        $ 646 "subir≔pose_sub(get_actual_tcp_pose(), bajada_broca)"
        global subir= pose_sub ( get_actual_tcp_pose (), bajada_broca)
        $ 647 "subir" "breakAfter"
        movel(subir, a=0.01, v=0.005)
        $ 648 "bajada_broca≔pose_sub(bajada_broca, bajada)"
        global bajada_broca= pose_sub (bajada_broca, bajada)
        Loop_42 = Loop_42 + 1
      end
      $ 649 "Direction: Base Z+"
      global move_thread_flag_649=0
      thread move_thread_649():
        enter_critical
        move_thread_flag_649 = 1
        local towardsPos=calculate_point_to_move_towards(p[0.0,0.0,0.0,0.0,0.0,0.0], [0.0,0.0,1.0], 0.06)
        movel(towardsPos, a=0.035, v=0.03)
        move_thread_flag_649 = 2
        exit_critical
      end
      move_thread_flag_649 = 0
      move_thread_han_649 = run move_thread_649()
      while (True):
        sleep(1.0E-10)
        if (move_thread_flag_649 > 1):
          join move_thread_han_649
          $ 650 "Until (distance)"
          break
        end
        sync()
      end
      $ 651 "Set CO[1]=Apagar"
      set_configurable_digital_out(1, False)
      $ 652 "barreno_actual≔barreno_actual+1"
      global barreno_actual=barreno_actual+1
      $ 653 "Call Quitar_broca"
      Quitar_broca()
      $ 654 "Call Poner_broca"
      Poner_broca()
    end
    $ 655 "EF"
    $ 656 "'desbaste_inicial'"
    # 'desbaste_inicial'
    $ 657 "bajada_broca≔p[0,0,-0.012,0,0,0]"
    global bajada_broca=p[0,0,-0.012,0,0,0]
    $ 658 "barrenos_menos1≔9"
    global barrenos_menos1=9
    $ 659 "barreno_actual≔0"
    global barreno_actual=0
    $ 660 "Loop barreno_actual≤barrenos_menos1"
    while (barreno_actual <= barrenos_menos1):
      $ 661 "Perforacion"
      $ 662 "MoveL"
      $ 663 "internos≔interpolate_pose(Linea2_E, Linea2_F, barreno_actual/barrenos_menos1)"
      global internos= interpolate_pose (Linea2_E_p, Linea2_F_p, barreno_actual/barrenos_menos1)
      $ 664 "internos" "breakAfter"
      movel(internos, a=0.5, v=0.1)
      $ 665 "'desbaste_inicial'"
      # 'desbaste_inicial'
      $ 666 "bajada_broca≔p[0,0,-0.012,0,0,0]"
      global bajada_broca=p[0,0,-0.012,0,0,0]
      $ 667 "bajada≔p[0,0,0.012,0,0,0]"
      global bajada=p[0,0,0.012,0,0,0]
      $ 668 "Direction: Base Z-"
      global move_thread_flag_668=0
      thread move_thread_668():
        enter_critical
        move_thread_flag_668 = 1
        local towardsPos=calculate_point_to_move_towards(p[0.0,0.0,0.0,0.0,0.0,0.0], [0.0,0.0,-1.0], 0.055)
        movel(towardsPos, a=0.025, v=0.02)
        move_thread_flag_668 = 2
        exit_critical
      end
      move_thread_flag_668 = 0
      move_thread_han_668 = run move_thread_668()
      while (True):
        sleep(1.0E-10)
        if (move_thread_flag_668 > 1):
          join move_thread_han_668
          $ 669 "Until (distance)"
          break
        end
        sync()
      end
      $ 670 "Popup: punto contacto alanzdo"
      popup("punto contacto alanzdo", "Mensaje", False, False, blocking=True)
      $ 671 "Direction: Base Z+"
      global move_thread_flag_671=0
      thread move_thread_671():
        enter_critical
        move_thread_flag_671 = 1
        local towardsPos=calculate_point_to_move_towards(p[0.0,0.0,0.0,0.0,0.0,0.0], [0.0,0.0,1.0], 0.001)
        movel(towardsPos, a=0.005, v=0.003)
        move_thread_flag_671 = 2
        exit_critical
      end
      move_thread_flag_671 = 0
      move_thread_han_671 = run move_thread_671()
      while (True):
        sleep(1.0E-10)
        if (move_thread_flag_671 > 1):
          join move_thread_han_671
          $ 672 "Until (distance)"
          break
        end
        sync()
      end
      $ 673 "Wait: 0.3"
      sleep(0.3)
      $ 674 "Set CO[1]=Encender"
      set_configurable_digital_out(1, True)
      $ 675 "Wait: 0.3"
      sleep(0.3)
      $ 676 "Loop 2 times"
      Loop_44 = 0
      while (Loop_44 < 2):
        $ 677 "bajar≔pose_add(get_actual_tcp_pose(), bajada_broca)"
        global bajar= pose_add ( get_actual_tcp_pose (), bajada_broca)
        $ 678 "bajar" "breakAfter"
        movel(bajar, a=0.005, v=0.001)
        $ 679 "subir≔pose_sub(get_actual_tcp_pose(), bajada_broca)"
        global subir= pose_sub ( get_actual_tcp_pose (), bajada_broca)
        $ 680 "subir" "breakAfter"
        movel(subir, a=0.01, v=0.005)
        $ 681 "bajada_broca≔pose_sub(bajada_broca, bajada)"
        global bajada_broca= pose_sub (bajada_broca, bajada)
        Loop_44 = Loop_44 + 1
      end
      $ 682 "Direction: Base Z+"
      global move_thread_flag_682=0
      thread move_thread_682():
        enter_critical
        move_thread_flag_682 = 1
        local towardsPos=calculate_point_to_move_towards(p[0.0,0.0,0.0,0.0,0.0,0.0], [0.0,0.0,1.0], 0.06)
        movel(towardsPos, a=0.035, v=0.03)
        move_thread_flag_682 = 2
        exit_critical
      end
      move_thread_flag_682 = 0
      move_thread_han_682 = run move_thread_682()
      while (True):
        sleep(1.0E-10)
        if (move_thread_flag_682 > 1):
          join move_thread_han_682
          $ 683 "Until (distance)"
          break
        end
        sync()
      end
      $ 684 "Set CO[1]=Apagar"
      set_configurable_digital_out(1, False)
      $ 685 "barreno_actual≔barreno_actual+1"
      global barreno_actual=barreno_actual+1
      $ 686 "If barreno_actual>barrenos_menos1"
      if (barreno_actual>barrenos_menos1):
        $ 687 "cambiar_broca≔ True "
        global cambiar_broca=  True
      end
      $ 688 "Call Quitar_broca"
      Quitar_broca()
      $ 689 "Call Poner_broca"
      Poner_broca()
    end
    $ 690 "Popup: Linea2 con full Terminada!"
    popup("Linea2 con full Terminada!", "Mensaje", False, False, blocking=True)
    $ 691 "Posicion3"
    $ 692 "eje7≔3"
    global eje7=3
    $ 693 "Broca_1"
    $ 694 "Linea3"
    $ 695 "Marcar_puntos"
    $ 696 "MoveL"
    $ 697 "punto_inicio1" "breakAfter"
    movel(punto_inicio1_p, a=0.5, v=0.1)
    $ 698 "Linea3_A" "breakAfter"
    movel(Linea3_A_p, a=0.5, v=0.1)
    $ 699 "Linea3_B" "breakAfter"
    movel(Linea3_B_p, a=0.5, v=0.1)
    $ 700 "Linea3_C" "breakAfter"
    movel(Linea3_C_p, a=0.5, v=0.1)
    $ 701 "Linea3_D" "breakAfter"
    movel(Linea3_D_p, a=0.5, v=0.1)
    $ 702 "Linea3_E" "breakAfter"
    movel(Linea3_E_p, a=0.5, v=0.1)
    $ 703 "Linea3_F" "breakAfter"
    movel(Linea3_F_p, a=0.5, v=0.1)
    $ 704 "AB"
    $ 705 "'desbaste_inicial'"
    # 'desbaste_inicial'
    $ 706 "bajada_broca≔p[0,0,-0.008,0,0,0]"
    global bajada_broca=p[0,0,-0.008,0,0,0]
    $ 707 "barrenos_menos1≔8"
    global barrenos_menos1=8
    $ 708 "barreno_actual≔0"
    global barreno_actual=0
    $ 709 "Loop barreno_actual≤barrenos_menos1"
    while (barreno_actual <= barrenos_menos1):
      $ 710 "Perforacion"
      $ 711 "MoveL"
      $ 712 "internos≔interpolate_pose(Linea3_A, Linea3_B, barreno_actual/barrenos_menos1)"
      global internos= interpolate_pose (Linea3_A_p, Linea3_B_p, barreno_actual/barrenos_menos1)
      $ 713 "internos" "breakAfter"
      movel(internos, a=0.5, v=0.1)
      $ 714 "'desbaste_inicial'"
      # 'desbaste_inicial'
      $ 715 "bajada_broca≔p[0,0,-0.008,0,0,0]"
      global bajada_broca=p[0,0,-0.008,0,0,0]
      $ 716 "bajada≔p[0,0,0.008,0,0,0]"
      global bajada=p[0,0,0.008,0,0,0]
      $ 717 "Direction: Base Z-"
      global move_thread_flag_717=0
      thread move_thread_717():
        enter_critical
        move_thread_flag_717 = 1
        local towardsPos=calculate_point_to_move_towards(p[0.0,0.0,0.0,0.0,0.0,0.0], [0.0,0.0,-1.0], 0.055)
        movel(towardsPos, a=0.015, v=0.02)
        move_thread_flag_717 = 2
        exit_critical
      end
      move_thread_flag_717 = 0
      move_thread_han_717 = run move_thread_717()
      while (True):
        sleep(1.0E-10)
        if (move_thread_flag_717 > 1):
          join move_thread_han_717
          $ 718 "Until (distance)"
          break
        end
        sync()
      end
      $ 719 "Popup: punto contacto alanzdo"
      popup("punto contacto alanzdo", "Mensaje", False, False, blocking=True)
      $ 720 "Direction: Base Z+"
      global move_thread_flag_720=0
      thread move_thread_720():
        enter_critical
        move_thread_flag_720 = 1
        local towardsPos=calculate_point_to_move_towards(p[0.0,0.0,0.0,0.0,0.0,0.0], [0.0,0.0,1.0], 0.001)
        movel(towardsPos, a=0.005, v=0.003)
        move_thread_flag_720 = 2
        exit_critical
      end
      move_thread_flag_720 = 0
      move_thread_han_720 = run move_thread_720()
      while (True):
        sleep(1.0E-10)
        if (move_thread_flag_720 > 1):
          join move_thread_han_720
          $ 721 "Until (distance)"
          break
        end
        sync()
      end
      $ 722 "Wait: 0.3"
      sleep(0.3)
      $ 723 "Set CO[1]=Encender"
      set_configurable_digital_out(1, True)
      $ 724 "Wait: 0.3"
      sleep(0.3)
      $ 725 "Loop 3 times"
      Loop_26 = 0
      while (Loop_26 < 3):
        $ 726 "bajar≔pose_add(get_actual_tcp_pose(), bajada_broca)"
        global bajar= pose_add ( get_actual_tcp_pose (), bajada_broca)
        $ 727 "bajar" "breakAfter"
        movel(bajar, a=0.005, v=0.001)
        $ 728 "subir≔pose_sub(get_actual_tcp_pose(), bajada_broca)"
        global subir= pose_sub ( get_actual_tcp_pose (), bajada_broca)
        $ 729 "subir" "breakAfter"
        movel(subir, a=0.01, v=0.005)
        $ 730 "bajada_broca≔pose_sub(bajada_broca, bajada)"
        global bajada_broca= pose_sub (bajada_broca, bajada)
        Loop_26 = Loop_26 + 1
      end
      $ 731 "Direction: Base Z+"
      global move_thread_flag_731=0
      thread move_thread_731():
        enter_critical
        move_thread_flag_731 = 1
        local towardsPos=calculate_point_to_move_towards(p[0.0,0.0,0.0,0.0,0.0,0.0], [0.0,0.0,1.0], 0.06)
        movel(towardsPos, a=0.035, v=0.03)
        move_thread_flag_731 = 2
        exit_critical
      end
      move_thread_flag_731 = 0
      move_thread_han_731 = run move_thread_731()
      while (True):
        sleep(1.0E-10)
        if (move_thread_flag_731 > 1):
          join move_thread_han_731
          $ 732 "Until (distance)"
          break
        end
        sync()
      end
      $ 733 "Set CO[1]=Apagar"
      set_configurable_digital_out(1, False)
      $ 734 "barreno_actual≔barreno_actual+1"
      global barreno_actual=barreno_actual+1
      $ 735 "Call Quitar_broca"
      Quitar_broca()
      $ 736 "Call Poner_broca"
      Poner_broca()
    end
    $ 737 "CD"
    $ 738 "'desbaste_inicial'"
    # 'desbaste_inicial'
    $ 739 "bajada_broca≔p[0,0,-0.008,0,0,0]"
    global bajada_broca=p[0,0,-0.008,0,0,0]
    $ 740 "barrenos_menos1≔8"
    global barrenos_menos1=8
    $ 741 "barreno_actual≔0"
    global barreno_actual=0
    $ 742 "Loop barreno_actual≤barrenos_menos1"
    while (barreno_actual <= barrenos_menos1):
      $ 743 "Perforacion"
      $ 744 "MoveL"
      $ 745 "internos≔interpolate_pose(Linea3_C, Linea3_D, barreno_actual/barrenos_menos1)"
      global internos= interpolate_pose (Linea3_C_p, Linea3_D_p, barreno_actual/barrenos_menos1)
      $ 746 "internos" "breakAfter"
      movel(internos, a=0.5, v=0.1)
      $ 747 "'desbaste_inicial'"
      # 'desbaste_inicial'
      $ 748 "bajada_broca≔p[0,0,-0.008,0,0,0]"
      global bajada_broca=p[0,0,-0.008,0,0,0]
      $ 749 "bajada≔p[0,0,0.008,0,0,0]"
      global bajada=p[0,0,0.008,0,0,0]
      $ 750 "Direction: Base Z-"
      global move_thread_flag_750=0
      thread move_thread_750():
        enter_critical
        move_thread_flag_750 = 1
        local towardsPos=calculate_point_to_move_towards(p[0.0,0.0,0.0,0.0,0.0,0.0], [0.0,0.0,-1.0], 0.055)
        movel(towardsPos, a=0.02, v=0.015)
        move_thread_flag_750 = 2
        exit_critical
      end
      move_thread_flag_750 = 0
      move_thread_han_750 = run move_thread_750()
      while (True):
        sleep(1.0E-10)
        if (move_thread_flag_750 > 1):
          join move_thread_han_750
          $ 751 "Until (distance)"
          break
        end
        sync()
      end
      $ 752 "Popup: punto contacto alanzdo"
      popup("punto contacto alanzdo", "Mensaje", False, False, blocking=True)
      $ 753 "Direction: Base Z+"
      global move_thread_flag_753=0
      thread move_thread_753():
        enter_critical
        move_thread_flag_753 = 1
        local towardsPos=calculate_point_to_move_towards(p[0.0,0.0,0.0,0.0,0.0,0.0], [0.0,0.0,1.0], 0.001)
        movel(towardsPos, a=0.005, v=0.003)
        move_thread_flag_753 = 2
        exit_critical
      end
      move_thread_flag_753 = 0
      move_thread_han_753 = run move_thread_753()
      while (True):
        sleep(1.0E-10)
        if (move_thread_flag_753 > 1):
          join move_thread_han_753
          $ 754 "Until (distance)"
          break
        end
        sync()
      end
      $ 755 "Wait: 0.3"
      sleep(0.3)
      $ 756 "Set CO[1]=Encender"
      set_configurable_digital_out(1, True)
      $ 757 "Wait: 0.3"
      sleep(0.3)
      $ 758 "Loop 3 times"
      Loop_28 = 0
      while (Loop_28 < 3):
        $ 759 "bajar≔pose_add(get_actual_tcp_pose(), bajada_broca)"
        global bajar= pose_add ( get_actual_tcp_pose (), bajada_broca)
        $ 760 "bajar" "breakAfter"
        movel(bajar, a=0.005, v=0.001)
        $ 761 "subir≔pose_sub(get_actual_tcp_pose(), bajada_broca)"
        global subir= pose_sub ( get_actual_tcp_pose (), bajada_broca)
        $ 762 "subir" "breakAfter"
        movel(subir, a=0.01, v=0.005)
        $ 763 "bajada_broca≔pose_sub(bajada_broca, bajada)"
        global bajada_broca= pose_sub (bajada_broca, bajada)
        Loop_28 = Loop_28 + 1
      end
      $ 764 "Direction: Base Z+"
      global move_thread_flag_764=0
      thread move_thread_764():
        enter_critical
        move_thread_flag_764 = 1
        local towardsPos=calculate_point_to_move_towards(p[0.0,0.0,0.0,0.0,0.0,0.0], [0.0,0.0,1.0], 0.06)
        movel(towardsPos, a=0.035, v=0.03)
        move_thread_flag_764 = 2
        exit_critical
      end
      move_thread_flag_764 = 0
      move_thread_han_764 = run move_thread_764()
      while (True):
        sleep(1.0E-10)
        if (move_thread_flag_764 > 1):
          join move_thread_han_764
          $ 765 "Until (distance)"
          break
        end
        sync()
      end
      $ 766 "Set CO[1]=Apagar"
      set_configurable_digital_out(1, False)
      $ 767 "barreno_actual≔barreno_actual+1"
      global barreno_actual=barreno_actual+1
      $ 768 "Call Quitar_broca"
      Quitar_broca()
      $ 769 "Call Poner_broca"
      Poner_broca()
    end
    $ 770 "EF"
    $ 771 "'desbaste_inicial'"
    # 'desbaste_inicial'
    $ 772 "bajada_broca≔p[0,0,-0.008,0,0,0]"
    global bajada_broca=p[0,0,-0.008,0,0,0]
    $ 773 "barrenos_menos1≔9"
    global barrenos_menos1=9
    $ 774 "barreno_actual≔0"
    global barreno_actual=0
    $ 775 "Loop barreno_actual≤barrenos_menos1"
    while (barreno_actual <= barrenos_menos1):
      $ 776 "Perforacion"
      $ 777 "MoveL"
      $ 778 "internos≔interpolate_pose(Linea3_E, Linea3_F, barreno_actual/barrenos_menos1)"
      global internos= interpolate_pose (Linea3_E_p, Linea3_F_p, barreno_actual/barrenos_menos1)
      $ 779 "internos" "breakAfter"
      movel(internos, a=0.5, v=0.1)
      $ 780 "'desbaste_inicial'"
      # 'desbaste_inicial'
      $ 781 "bajada_broca≔p[0,0,-0.008,0,0,0]"
      global bajada_broca=p[0,0,-0.008,0,0,0]
      $ 782 "bajada≔p[0,0,0.008,0,0,0]"
      global bajada=p[0,0,0.008,0,0,0]
      $ 783 "Direction: Base Z-"
      global move_thread_flag_783=0
      thread move_thread_783():
        enter_critical
        move_thread_flag_783 = 1
        local towardsPos=calculate_point_to_move_towards(p[0.0,0.0,0.0,0.0,0.0,0.0], [0.0,0.0,-1.0], 0.055)
        movel(towardsPos, a=0.015, v=0.02)
        move_thread_flag_783 = 2
        exit_critical
      end
      move_thread_flag_783 = 0
      move_thread_han_783 = run move_thread_783()
      while (True):
        sleep(1.0E-10)
        if (move_thread_flag_783 > 1):
          join move_thread_han_783
          $ 784 "Until (distance)"
          break
        end
        sync()
      end
      $ 785 "Popup: punto contacto alanzdo"
      popup("punto contacto alanzdo", "Mensaje", False, False, blocking=True)
      $ 786 "Direction: Base Z+"
      global move_thread_flag_786=0
      thread move_thread_786():
        enter_critical
        move_thread_flag_786 = 1
        local towardsPos=calculate_point_to_move_towards(p[0.0,0.0,0.0,0.0,0.0,0.0], [0.0,0.0,1.0], 0.001)
        movel(towardsPos, a=0.005, v=0.003)
        move_thread_flag_786 = 2
        exit_critical
      end
      move_thread_flag_786 = 0
      move_thread_han_786 = run move_thread_786()
      while (True):
        sleep(1.0E-10)
        if (move_thread_flag_786 > 1):
          join move_thread_han_786
          $ 787 "Until (distance)"
          break
        end
        sync()
      end
      $ 788 "Wait: 0.3"
      sleep(0.3)
      $ 789 "Set CO[1]=Encender"
      set_configurable_digital_out(1, True)
      $ 790 "Wait: 0.3"
      sleep(0.3)
      $ 791 "Loop 3 times"
      Loop_30 = 0
      while (Loop_30 < 3):
        $ 792 "bajar≔pose_add(get_actual_tcp_pose(), bajada_broca)"
        global bajar= pose_add ( get_actual_tcp_pose (), bajada_broca)
        $ 793 "bajar" "breakAfter"
        movel(bajar, a=0.005, v=0.001)
        $ 794 "subir≔pose_sub(get_actual_tcp_pose(), bajada_broca)"
        global subir= pose_sub ( get_actual_tcp_pose (), bajada_broca)
        $ 795 "subir" "breakAfter"
        movel(subir, a=0.01, v=0.005)
        $ 796 "bajada_broca≔pose_sub(bajada_broca, bajada)"
        global bajada_broca= pose_sub (bajada_broca, bajada)
        Loop_30 = Loop_30 + 1
      end
      $ 797 "Direction: Base Z+"
      global move_thread_flag_797=0
      thread move_thread_797():
        enter_critical
        move_thread_flag_797 = 1
        local towardsPos=calculate_point_to_move_towards(p[0.0,0.0,0.0,0.0,0.0,0.0], [0.0,0.0,1.0], 0.06)
        movel(towardsPos, a=0.035, v=0.03)
        move_thread_flag_797 = 2
        exit_critical
      end
      move_thread_flag_797 = 0
      move_thread_han_797 = run move_thread_797()
      while (True):
        sleep(1.0E-10)
        if (move_thread_flag_797 > 1):
          join move_thread_han_797
          $ 798 "Until (distance)"
          break
        end
        sync()
      end
      $ 799 "Set CO[1]=Apagar"
      set_configurable_digital_out(1, False)
      $ 800 "barreno_actual≔barreno_actual+1"
      global barreno_actual=barreno_actual+1
      $ 801 "Call Quitar_broca"
      Quitar_broca()
      $ 802 "Call Poner_broca"
      Poner_broca()
    end
    $ 803 "Popup: Linea1 con chica Terminada!"
    popup("Linea1 con chica Terminada!", "Mensaje", False, False, blocking=True)
    $ 804 "Linea4"
    $ 805 "Marcar_puntos"
    $ 806 "MoveL"
    $ 807 "punto_inicio1" "breakAfter"
    movel(punto_inicio1_p, a=0.5, v=0.1)
    $ 808 "Linea4_A" "breakAfter"
    movel(Linea4_A_p, a=0.5, v=0.1)
    $ 809 "Linea4_B" "breakAfter"
    movel(Linea4_B_p, a=0.5, v=0.1)
    $ 810 "Linea4_C" "breakAfter"
    movel(Linea4_C_p, a=0.5, v=0.1)
    $ 811 "Linea4_D" "breakAfter"
    movel(Linea4_D_p, a=0.5, v=0.1)
    $ 812 "Linea4_E" "breakAfter"
    movel(Linea4_E_p, a=0.5, v=0.1)
    $ 813 "Linea4_F" "breakAfter"
    movel(Linea4_F_p, a=0.5, v=0.1)
    $ 814 "AB"
    $ 815 "'desbaste_inicial'"
    # 'desbaste_inicial'
    $ 816 "bajada_broca≔p[0,0,-0.008,0,0,0]"
    global bajada_broca=p[0,0,-0.008,0,0,0]
    $ 817 "barrenos_menos1≔8"
    global barrenos_menos1=8
    $ 818 "barreno_actual≔0"
    global barreno_actual=0
    $ 819 "Loop barreno_actual≤barrenos_menos1"
    while (barreno_actual <= barrenos_menos1):
      $ 820 "Perforacion"
      $ 821 "MoveL"
      $ 822 "internos≔interpolate_pose(Linea4_A, Linea4_B, barreno_actual/barrenos_menos1)"
      global internos= interpolate_pose (Linea4_A_p, Linea4_B_p, barreno_actual/barrenos_menos1)
      $ 823 "internos" "breakAfter"
      movel(internos, a=0.5, v=0.1)
      $ 824 "'desbaste_inicial'"
      # 'desbaste_inicial'
      $ 825 "bajada_broca≔p[0,0,-0.008,0,0,0]"
      global bajada_broca=p[0,0,-0.008,0,0,0]
      $ 826 "bajada≔p[0,0,0.008,0,0,0]"
      global bajada=p[0,0,0.008,0,0,0]
      $ 827 "Direction: Base Z-"
      global move_thread_flag_827=0
      thread move_thread_827():
        enter_critical
        move_thread_flag_827 = 1
        local towardsPos=calculate_point_to_move_towards(p[0.0,0.0,0.0,0.0,0.0,0.0], [0.0,0.0,-1.0], 0.055)
        movel(towardsPos, a=0.015, v=0.02)
        move_thread_flag_827 = 2
        exit_critical
      end
      move_thread_flag_827 = 0
      move_thread_han_827 = run move_thread_827()
      while (True):
        sleep(1.0E-10)
        if (move_thread_flag_827 > 1):
          join move_thread_han_827
          $ 828 "Until (distance)"
          break
        end
        sync()
      end
      $ 829 "Popup: punto contacto alanzdo"
      popup("punto contacto alanzdo", "Mensaje", False, False, blocking=True)
      $ 830 "Direction: Base Z+"
      global move_thread_flag_830=0
      thread move_thread_830():
        enter_critical
        move_thread_flag_830 = 1
        local towardsPos=calculate_point_to_move_towards(p[0.0,0.0,0.0,0.0,0.0,0.0], [0.0,0.0,1.0], 0.002)
        movel(towardsPos, a=0.005, v=0.003)
        move_thread_flag_830 = 2
        exit_critical
      end
      move_thread_flag_830 = 0
      move_thread_han_830 = run move_thread_830()
      while (True):
        sleep(1.0E-10)
        if (move_thread_flag_830 > 1):
          join move_thread_han_830
          $ 831 "Until (distance)"
          break
        end
        sync()
      end
      $ 832 "Wait: 0.3"
      sleep(0.3)
      $ 833 "Set CO[1]=Encender"
      set_configurable_digital_out(1, True)
      $ 834 "Wait: 0.3"
      sleep(0.3)
      $ 835 "Loop 3 times"
      Loop_32 = 0
      while (Loop_32 < 3):
        $ 836 "bajar≔pose_add(get_actual_tcp_pose(), bajada_broca)"
        global bajar= pose_add ( get_actual_tcp_pose (), bajada_broca)
        $ 837 "bajar" "breakAfter"
        movel(bajar, a=0.005, v=0.001)
        $ 838 "subir≔pose_sub(get_actual_tcp_pose(), bajada_broca)"
        global subir= pose_sub ( get_actual_tcp_pose (), bajada_broca)
        $ 839 "subir" "breakAfter"
        movel(subir, a=0.01, v=0.005)
        $ 840 "bajada_broca≔pose_sub(bajada_broca, bajada)"
        global bajada_broca= pose_sub (bajada_broca, bajada)
        Loop_32 = Loop_32 + 1
      end
      $ 841 "Direction: Base Z+"
      global move_thread_flag_841=0
      thread move_thread_841():
        enter_critical
        move_thread_flag_841 = 1
        local towardsPos=calculate_point_to_move_towards(p[0.0,0.0,0.0,0.0,0.0,0.0], [0.0,0.0,1.0], 0.06)
        movel(towardsPos, a=0.035, v=0.03)
        move_thread_flag_841 = 2
        exit_critical
      end
      move_thread_flag_841 = 0
      move_thread_han_841 = run move_thread_841()
      while (True):
        sleep(1.0E-10)
        if (move_thread_flag_841 > 1):
          join move_thread_han_841
          $ 842 "Until (distance)"
          break
        end
        sync()
      end
      $ 843 "Set CO[1]=Apagar"
      set_configurable_digital_out(1, False)
      $ 844 "barreno_actual≔barreno_actual+1"
      global barreno_actual=barreno_actual+1
    end
    $ 847 "CD"
    $ 848 "'desbaste_inicial'"
    # 'desbaste_inicial'
    $ 849 "bajada_broca≔p[0,0,-0.008,0,0,0]"
    global bajada_broca=p[0,0,-0.008,0,0,0]
    $ 850 "barrenos_menos1≔8"
    global barrenos_menos1=8
    $ 851 "barreno_actual≔0"
    global barreno_actual=0
    $ 852 "Loop barreno_actual≤barrenos_menos1"
    while (barreno_actual <= barrenos_menos1):
      $ 853 "Perforacion"
      $ 854 "MoveL"
      $ 855 "internos≔interpolate_pose(Linea4_C, Linea4_D, barreno_actual/barrenos_menos1)"
      global internos= interpolate_pose (Linea4_C_p, Linea4_D_p, barreno_actual/barrenos_menos1)
      $ 856 "internos" "breakAfter"
      movel(internos, a=0.5, v=0.1)
      $ 857 "'desbaste_inicial'"
      # 'desbaste_inicial'
      $ 858 "bajada_broca≔p[0,0,-0.008,0,0,0]"
      global bajada_broca=p[0,0,-0.008,0,0,0]
      $ 859 "bajada≔p[0,0,0.008,0,0,0]"
      global bajada=p[0,0,0.008,0,0,0]
      $ 860 "Direction: Base Z-"
      global move_thread_flag_860=0
      thread move_thread_860():
        enter_critical
        move_thread_flag_860 = 1
        local towardsPos=calculate_point_to_move_towards(p[0.0,0.0,0.0,0.0,0.0,0.0], [0.0,0.0,-1.0], 0.055)
        movel(towardsPos, a=0.015, v=0.02)
        move_thread_flag_860 = 2
        exit_critical
      end
      move_thread_flag_860 = 0
      move_thread_han_860 = run move_thread_860()
      while (True):
        sleep(1.0E-10)
        if (move_thread_flag_860 > 1):
          join move_thread_han_860
          $ 861 "Until (distance)"
          break
        end
        sync()
      end
      $ 862 "Popup: punto contacto alanzdo"
      popup("punto contacto alanzdo", "Mensaje", False, False, blocking=True)
      $ 863 "Direction: Base Z+"
      global move_thread_flag_863=0
      thread move_thread_863():
        enter_critical
        move_thread_flag_863 = 1
        local towardsPos=calculate_point_to_move_towards(p[0.0,0.0,0.0,0.0,0.0,0.0], [0.0,0.0,1.0], 0.002)
        movel(towardsPos, a=0.005, v=0.003)
        move_thread_flag_863 = 2
        exit_critical
      end
      move_thread_flag_863 = 0
      move_thread_han_863 = run move_thread_863()
      while (True):
        sleep(1.0E-10)
        if (move_thread_flag_863 > 1):
          join move_thread_han_863
          $ 864 "Until (distance)"
          break
        end
        sync()
      end
      $ 865 "Wait: 0.3"
      sleep(0.3)
      $ 866 "Set CO[1]=Encender"
      set_configurable_digital_out(1, True)
      $ 867 "Wait: 0.3"
      sleep(0.3)
      $ 868 "Loop 3 times"
      Loop_35 = 0
      while (Loop_35 < 3):
        $ 869 "bajar≔pose_add(get_actual_tcp_pose(), bajada_broca)"
        global bajar= pose_add ( get_actual_tcp_pose (), bajada_broca)
        $ 870 "bajar" "breakAfter"
        movel(bajar, a=0.005, v=0.001)
        $ 871 "subir≔pose_sub(get_actual_tcp_pose(), bajada_broca)"
        global subir= pose_sub ( get_actual_tcp_pose (), bajada_broca)
        $ 872 "subir" "breakAfter"
        movel(subir, a=0.01, v=0.005)
        $ 873 "bajada_broca≔pose_sub(bajada_broca, bajada)"
        global bajada_broca= pose_sub (bajada_broca, bajada)
        Loop_35 = Loop_35 + 1
      end
      $ 874 "Direction: Base Z+"
      global move_thread_flag_874=0
      thread move_thread_874():
        enter_critical
        move_thread_flag_874 = 1
        local towardsPos=calculate_point_to_move_towards(p[0.0,0.0,0.0,0.0,0.0,0.0], [0.0,0.0,1.0], 0.06)
        movel(towardsPos, a=0.035, v=0.03)
        move_thread_flag_874 = 2
        exit_critical
      end
      move_thread_flag_874 = 0
      move_thread_han_874 = run move_thread_874()
      while (True):
        sleep(1.0E-10)
        if (move_thread_flag_874 > 1):
          join move_thread_han_874
          $ 875 "Until (distance)"
          break
        end
        sync()
      end
      $ 876 "Set CO[1]=Apagar"
      set_configurable_digital_out(1, False)
      $ 877 "barreno_actual≔barreno_actual+1"
      global barreno_actual=barreno_actual+1
    end
    $ 880 "EF"
    $ 881 "'desbaste_inicial'"
    # 'desbaste_inicial'
    $ 882 "bajada_broca≔p[0,0,-0.008,0,0,0]"
    global bajada_broca=p[0,0,-0.008,0,0,0]
    $ 883 "barrenos_menos1≔9"
    global barrenos_menos1=9
    $ 884 "barreno_actual≔0"
    global barreno_actual=0
    $ 885 "Loop barreno_actual≤barrenos_menos1"
    while (barreno_actual <= barrenos_menos1):
      $ 886 "Perforacion"
      $ 887 "MoveL"
      $ 888 "internos≔interpolate_pose(Linea4_E, Linea4_F, barreno_actual/barrenos_menos1)"
      global internos= interpolate_pose (Linea4_E_p, Linea4_F_p, barreno_actual/barrenos_menos1)
      $ 889 "internos" "breakAfter"
      movel(internos, a=0.5, v=0.1)
      $ 890 "'desbaste_inicial'"
      # 'desbaste_inicial'
      $ 891 "bajada_broca≔p[0,0,-0.008,0,0,0]"
      global bajada_broca=p[0,0,-0.008,0,0,0]
      $ 892 "bajada≔p[0,0,0.008,0,0,0]"
      global bajada=p[0,0,0.008,0,0,0]
      $ 893 "Direction: Base Z-"
      global move_thread_flag_893=0
      thread move_thread_893():
        enter_critical
        move_thread_flag_893 = 1
        local towardsPos=calculate_point_to_move_towards(p[0.0,0.0,0.0,0.0,0.0,0.0], [0.0,0.0,-1.0], 0.055)
        movel(towardsPos, a=0.015, v=0.02)
        move_thread_flag_893 = 2
        exit_critical
      end
      move_thread_flag_893 = 0
      move_thread_han_893 = run move_thread_893()
      while (True):
        sleep(1.0E-10)
        if (move_thread_flag_893 > 1):
          join move_thread_han_893
          $ 894 "Until (distance)"
          break
        end
        sync()
      end
      $ 895 "Popup: punto contacto alanzdo"
      popup("punto contacto alanzdo", "Mensaje", False, False, blocking=True)
      $ 896 "Direction: Base Z+"
      global move_thread_flag_896=0
      thread move_thread_896():
        enter_critical
        move_thread_flag_896 = 1
        local towardsPos=calculate_point_to_move_towards(p[0.0,0.0,0.0,0.0,0.0,0.0], [0.0,0.0,1.0], 0.002)
        movel(towardsPos, a=0.005, v=0.003)
        move_thread_flag_896 = 2
        exit_critical
      end
      move_thread_flag_896 = 0
      move_thread_han_896 = run move_thread_896()
      while (True):
        sleep(1.0E-10)
        if (move_thread_flag_896 > 1):
          join move_thread_han_896
          $ 897 "Until (distance)"
          break
        end
        sync()
      end
      $ 898 "Wait: 0.3"
      sleep(0.3)
      $ 899 "Set CO[1]=Encender"
      set_configurable_digital_out(1, True)
      $ 900 "Wait: 0.3"
      sleep(0.3)
      $ 901 "Loop 3 times"
      Loop_39 = 0
      while (Loop_39 < 3):
        $ 902 "bajar≔pose_add(get_actual_tcp_pose(), bajada_broca)"
        global bajar= pose_add ( get_actual_tcp_pose (), bajada_broca)
        $ 903 "bajar" "breakAfter"
        movel(bajar, a=0.005, v=0.001)
        $ 904 "subir≔pose_sub(get_actual_tcp_pose(), bajada_broca)"
        global subir= pose_sub ( get_actual_tcp_pose (), bajada_broca)
        $ 905 "subir" "breakAfter"
        movel(subir, a=0.01, v=0.005)
        $ 906 "bajada_broca≔pose_sub(bajada_broca, bajada)"
        global bajada_broca= pose_sub (bajada_broca, bajada)
        Loop_39 = Loop_39 + 1
      end
      $ 907 "Direction: Base Z+"
      global move_thread_flag_907=0
      thread move_thread_907():
        enter_critical
        move_thread_flag_907 = 1
        local towardsPos=calculate_point_to_move_towards(p[0.0,0.0,0.0,0.0,0.0,0.0], [0.0,0.0,1.0], 0.06)
        movel(towardsPos, a=0.035, v=0.03)
        move_thread_flag_907 = 2
        exit_critical
      end
      move_thread_flag_907 = 0
      move_thread_han_907 = run move_thread_907()
      while (True):
        sleep(1.0E-10)
        if (move_thread_flag_907 > 1):
          join move_thread_han_907
          $ 908 "Until (distance)"
          break
        end
        sync()
      end
      $ 909 "Set CO[1]=Apagar"
      set_configurable_digital_out(1, False)
      $ 910 "barreno_actual≔barreno_actual+1"
      global barreno_actual=barreno_actual+1
      $ 911 "If barreno_actual>barrenos_menos1"
      if (barreno_actual>barrenos_menos1):
        $ 912 "cambiar_broca≔ True "
        global cambiar_broca=  True
      end
    end
    $ 915 "Popup: Linea2 con chica Terminada!"
    popup("Linea2 con chica Terminada!", "Mensaje", False, False, blocking=True)
    $ 916 "Broca_2"
    $ 917 "Linea3"
    $ 918 "Marcar_puntos"
    $ 919 "MoveL"
    $ 920 "punto_inicio1" "breakAfter"
    movel(punto_inicio1_p, a=0.5, v=0.1)
    $ 921 "Linea3_A" "breakAfter"
    movel(Linea3_A_p, a=0.5, v=0.1)
    $ 922 "Linea3_B" "breakAfter"
    movel(Linea3_B_p, a=0.5, v=0.1)
    $ 923 "Linea3_C" "breakAfter"
    movel(Linea3_C_p, a=0.5, v=0.1)
    $ 924 "Linea3_D" "breakAfter"
    movel(Linea3_D_p, a=0.5, v=0.1)
    $ 925 "Linea3_E" "breakAfter"
    movel(Linea3_E_p, a=0.5, v=0.1)
    $ 926 "Linea3_F" "breakAfter"
    movel(Linea3_F_p, a=0.5, v=0.1)
    $ 927 "AB"
    $ 928 "'desbaste_inicial'"
    # 'desbaste_inicial'
    $ 929 "bajada_broca≔p[0,0,-0.012,0,0,0]"
    global bajada_broca=p[0,0,-0.012,0,0,0]
    $ 930 "barrenos_menos1≔8"
    global barrenos_menos1=8
    $ 931 "barreno_actual≔0"
    global barreno_actual=0
    $ 932 "Loop barreno_actual≤barrenos_menos1"
    while (barreno_actual <= barrenos_menos1):
      $ 933 "Perforacion"
      $ 934 "MoveL"
      $ 935 "internos≔interpolate_pose(Linea3_A, Linea3_B, barreno_actual/barrenos_menos1)"
      global internos= interpolate_pose (Linea3_A_p, Linea3_B_p, barreno_actual/barrenos_menos1)
      $ 936 "internos" "breakAfter"
      movel(internos, a=0.5, v=0.1)
      $ 937 "'desbaste_inicial'"
      # 'desbaste_inicial'
      $ 938 "bajada_broca≔p[0,0,-0.012,0,0,0]"
      global bajada_broca=p[0,0,-0.012,0,0,0]
      $ 939 "bajada≔p[0,0,0.012,0,0,0]"
      global bajada=p[0,0,0.012,0,0,0]
      $ 940 "Direction: Base Z-"
      global move_thread_flag_940=0
      thread move_thread_940():
        enter_critical
        move_thread_flag_940 = 1
        local towardsPos=calculate_point_to_move_towards(p[0.0,0.0,0.0,0.0,0.0,0.0], [0.0,0.0,-1.0], 0.055)
        movel(towardsPos, a=0.015, v=0.02)
        move_thread_flag_940 = 2
        exit_critical
      end
      move_thread_flag_940 = 0
      move_thread_han_940 = run move_thread_940()
      while (True):
        sleep(1.0E-10)
        if (move_thread_flag_940 > 1):
          join move_thread_han_940
          $ 941 "Until (distance)"
          break
        end
        sync()
      end
      $ 942 "Popup: punto contacto alanzdo"
      popup("punto contacto alanzdo", "Mensaje", False, False, blocking=True)
      $ 943 "Direction: Base Z+"
      global move_thread_flag_943=0
      thread move_thread_943():
        enter_critical
        move_thread_flag_943 = 1
        local towardsPos=calculate_point_to_move_towards(p[0.0,0.0,0.0,0.0,0.0,0.0], [0.0,0.0,1.0], 0.002)
        movel(towardsPos, a=0.005, v=0.003)
        move_thread_flag_943 = 2
        exit_critical
      end
      move_thread_flag_943 = 0
      move_thread_han_943 = run move_thread_943()
      while (True):
        sleep(1.0E-10)
        if (move_thread_flag_943 > 1):
          join move_thread_han_943
          $ 944 "Until (distance)"
          break
        end
        sync()
      end
      $ 945 "Wait: 0.3"
      sleep(0.3)
      $ 946 "Set CO[1]=Encender"
      set_configurable_digital_out(1, True)
      $ 947 "Wait: 0.3"
      sleep(0.3)
      $ 948 "Loop 2 times"
      Loop_70 = 0
      while (Loop_70 < 2):
        $ 949 "bajar≔pose_add(get_actual_tcp_pose(), bajada_broca)"
        global bajar= pose_add ( get_actual_tcp_pose (), bajada_broca)
        $ 950 "bajar" "breakAfter"
        movel(bajar, a=0.005, v=0.001)
        $ 951 "subir≔pose_sub(get_actual_tcp_pose(), bajada_broca)"
        global subir= pose_sub ( get_actual_tcp_pose (), bajada_broca)
        $ 952 "subir" "breakAfter"
        movel(subir, a=0.01, v=0.005)
        $ 953 "bajada_broca≔pose_sub(bajada_broca, bajada)"
        global bajada_broca= pose_sub (bajada_broca, bajada)
        Loop_70 = Loop_70 + 1
      end
      $ 954 "Direction: Base Z+"
      global move_thread_flag_954=0
      thread move_thread_954():
        enter_critical
        move_thread_flag_954 = 1
        local towardsPos=calculate_point_to_move_towards(p[0.0,0.0,0.0,0.0,0.0,0.0], [0.0,0.0,1.0], 0.06)
        movel(towardsPos, a=0.035, v=0.03)
        move_thread_flag_954 = 2
        exit_critical
      end
      move_thread_flag_954 = 0
      move_thread_han_954 = run move_thread_954()
      while (True):
        sleep(1.0E-10)
        if (move_thread_flag_954 > 1):
          join move_thread_han_954
          $ 955 "Until (distance)"
          break
        end
        sync()
      end
      $ 956 "Set CO[1]=Apagar"
      set_configurable_digital_out(1, False)
      $ 957 "barreno_actual≔barreno_actual+1"
      global barreno_actual=barreno_actual+1
    end
    $ 960 "CD"
    $ 961 "'desbaste_inicial'"
    # 'desbaste_inicial'
    $ 962 "bajada_broca≔p[0,0,-0.012,0,0,0]"
    global bajada_broca=p[0,0,-0.012,0,0,0]
    $ 963 "barrenos_menos1≔8"
    global barrenos_menos1=8
    $ 964 "barreno_actual≔0"
    global barreno_actual=0
    $ 965 "Loop barreno_actual≤barrenos_menos1"
    while (barreno_actual <= barrenos_menos1):
      $ 966 "Perforacion"
      $ 967 "MoveL"
      $ 968 "internos≔interpolate_pose(Linea3_C, Linea3_D, barreno_actual/barrenos_menos1)"
      global internos= interpolate_pose (Linea3_C_p, Linea3_D_p, barreno_actual/barrenos_menos1)
      $ 969 "internos" "breakAfter"
      movel(internos, a=0.5, v=0.1)
      $ 970 "'desbaste_inicial'"
      # 'desbaste_inicial'
      $ 971 "bajada_broca≔p[0,0,-0.012,0,0,0]"
      global bajada_broca=p[0,0,-0.012,0,0,0]
      $ 972 "bajada≔p[0,0,0.012,0,0,0]"
      global bajada=p[0,0,0.012,0,0,0]
      $ 973 "Direction: Base Z-"
      global move_thread_flag_973=0
      thread move_thread_973():
        enter_critical
        move_thread_flag_973 = 1
        local towardsPos=calculate_point_to_move_towards(p[0.0,0.0,0.0,0.0,0.0,0.0], [0.0,0.0,-1.0], 0.055)
        movel(towardsPos, a=0.02, v=0.015)
        move_thread_flag_973 = 2
        exit_critical
      end
      move_thread_flag_973 = 0
      move_thread_han_973 = run move_thread_973()
      while (True):
        sleep(1.0E-10)
        if (move_thread_flag_973 > 1):
          join move_thread_han_973
          $ 974 "Until (distance)"
          break
        end
        sync()
      end
      $ 975 "Popup: punto contacto alanzdo"
      popup("punto contacto alanzdo", "Mensaje", False, False, blocking=True)
      $ 976 "Direction: Base Z+"
      global move_thread_flag_976=0
      thread move_thread_976():
        enter_critical
        move_thread_flag_976 = 1
        local towardsPos=calculate_point_to_move_towards(p[0.0,0.0,0.0,0.0,0.0,0.0], [0.0,0.0,1.0], 0.002)
        movel(towardsPos, a=0.005, v=0.003)
        move_thread_flag_976 = 2
        exit_critical
      end
      move_thread_flag_976 = 0
      move_thread_han_976 = run move_thread_976()
      while (True):
        sleep(1.0E-10)
        if (move_thread_flag_976 > 1):
          join move_thread_han_976
          $ 977 "Until (distance)"
          break
        end
        sync()
      end
      $ 978 "Wait: 0.3"
      sleep(0.3)
      $ 979 "Set CO[1]=Encender"
      set_configurable_digital_out(1, True)
      $ 980 "Wait: 0.3"
      sleep(0.3)
      $ 981 "Loop 2 times"
      Loop_72 = 0
      while (Loop_72 < 2):
        $ 982 "bajar≔pose_add(get_actual_tcp_pose(), bajada_broca)"
        global bajar= pose_add ( get_actual_tcp_pose (), bajada_broca)
        $ 983 "bajar" "breakAfter"
        movel(bajar, a=0.005, v=0.001)
        $ 984 "subir≔pose_sub(get_actual_tcp_pose(), bajada_broca)"
        global subir= pose_sub ( get_actual_tcp_pose (), bajada_broca)
        $ 985 "subir" "breakAfter"
        movel(subir, a=0.01, v=0.005)
        $ 986 "bajada_broca≔pose_sub(bajada_broca, bajada)"
        global bajada_broca= pose_sub (bajada_broca, bajada)
        Loop_72 = Loop_72 + 1
      end
      $ 987 "Direction: Base Z+"
      global move_thread_flag_987=0
      thread move_thread_987():
        enter_critical
        move_thread_flag_987 = 1
        local towardsPos=calculate_point_to_move_towards(p[0.0,0.0,0.0,0.0,0.0,0.0], [0.0,0.0,1.0], 0.06)
        movel(towardsPos, a=0.035, v=0.03)
        move_thread_flag_987 = 2
        exit_critical
      end
      move_thread_flag_987 = 0
      move_thread_han_987 = run move_thread_987()
      while (True):
        sleep(1.0E-10)
        if (move_thread_flag_987 > 1):
          join move_thread_han_987
          $ 988 "Until (distance)"
          break
        end
        sync()
      end
      $ 989 "Set CO[1]=Apagar"
      set_configurable_digital_out(1, False)
      $ 990 "barreno_actual≔barreno_actual+1"
      global barreno_actual=barreno_actual+1
    end
    $ 993 "EF"
    $ 994 "'desbaste_inicial'"
    # 'desbaste_inicial'
    $ 995 "bajada_broca≔p[0,0,-0.012,0,0,0]"
    global bajada_broca=p[0,0,-0.012,0,0,0]
    $ 996 "barrenos_menos1≔9"
    global barrenos_menos1=9
    $ 997 "barreno_actual≔0"
    global barreno_actual=0
    $ 998 "Loop barreno_actual≤barrenos_menos1"
    while (barreno_actual <= barrenos_menos1):
      $ 999 "Perforacion"
      $ 1000 "MoveL"
      $ 1001 "internos≔interpolate_pose(Linea3_E, Linea3_F, barreno_actual/barrenos_menos1)"
      global internos= interpolate_pose (Linea3_E_p, Linea3_F_p, barreno_actual/barrenos_menos1)
      $ 1002 "internos" "breakAfter"
      movel(internos, a=0.5, v=0.1)
      $ 1003 "'desbaste_inicial'"
      # 'desbaste_inicial'
      $ 1004 "bajada_broca≔p[0,0,-0.012,0,0,0]"
      global bajada_broca=p[0,0,-0.012,0,0,0]
      $ 1005 "bajada≔p[0,0,0.012,0,0,0]"
      global bajada=p[0,0,0.012,0,0,0]
      $ 1006 "Direction: Base Z-"
      global move_thread_flag_1006=0
      thread move_thread_1006():
        enter_critical
        move_thread_flag_1006 = 1
        local towardsPos=calculate_point_to_move_towards(p[0.0,0.0,0.0,0.0,0.0,0.0], [0.0,0.0,-1.0], 0.055)
        movel(towardsPos, a=0.015, v=0.02)
        move_thread_flag_1006 = 2
        exit_critical
      end
      move_thread_flag_1006 = 0
      move_thread_han_1006 = run move_thread_1006()
      while (True):
        sleep(1.0E-10)
        if (move_thread_flag_1006 > 1):
          join move_thread_han_1006
          $ 1007 "Until (distance)"
          break
        end
        sync()
      end
      $ 1008 "Popup: punto contacto alanzdo"
      popup("punto contacto alanzdo", "Mensaje", False, False, blocking=True)
      $ 1009 "Direction: Base Z+"
      global move_thread_flag_1009=0
      thread move_thread_1009():
        enter_critical
        move_thread_flag_1009 = 1
        local towardsPos=calculate_point_to_move_towards(p[0.0,0.0,0.0,0.0,0.0,0.0], [0.0,0.0,1.0], 0.002)
        movel(towardsPos, a=0.005, v=0.003)
        move_thread_flag_1009 = 2
        exit_critical
      end
      move_thread_flag_1009 = 0
      move_thread_han_1009 = run move_thread_1009()
      while (True):
        sleep(1.0E-10)
        if (move_thread_flag_1009 > 1):
          join move_thread_han_1009
          $ 1010 "Until (distance)"
          break
        end
        sync()
      end
      $ 1011 "Wait: 0.3"
      sleep(0.3)
      $ 1012 "Set CO[1]=Encender"
      set_configurable_digital_out(1, True)
      $ 1013 "Wait: 0.3"
      sleep(0.3)
      $ 1014 "Loop 2 times"
      Loop_74 = 0
      while (Loop_74 < 2):
        $ 1015 "bajar≔pose_add(get_actual_tcp_pose(), bajada_broca)"
        global bajar= pose_add ( get_actual_tcp_pose (), bajada_broca)
        $ 1016 "bajar" "breakAfter"
        movel(bajar, a=0.005, v=0.001)
        $ 1017 "subir≔pose_sub(get_actual_tcp_pose(), bajada_broca)"
        global subir= pose_sub ( get_actual_tcp_pose (), bajada_broca)
        $ 1018 "subir" "breakAfter"
        movel(subir, a=0.01, v=0.005)
        $ 1019 "bajada_broca≔pose_sub(bajada_broca, bajada)"
        global bajada_broca= pose_sub (bajada_broca, bajada)
        Loop_74 = Loop_74 + 1
      end
      $ 1020 "Direction: Base Z+"
      global move_thread_flag_1020=0
      thread move_thread_1020():
        enter_critical
        move_thread_flag_1020 = 1
        local towardsPos=calculate_point_to_move_towards(p[0.0,0.0,0.0,0.0,0.0,0.0], [0.0,0.0,1.0], 0.06)
        movel(towardsPos, a=0.035, v=0.03)
        move_thread_flag_1020 = 2
        exit_critical
      end
      move_thread_flag_1020 = 0
      move_thread_han_1020 = run move_thread_1020()
      while (True):
        sleep(1.0E-10)
        if (move_thread_flag_1020 > 1):
          join move_thread_han_1020
          $ 1021 "Until (distance)"
          break
        end
        sync()
      end
      $ 1022 "Set CO[1]=Apagar"
      set_configurable_digital_out(1, False)
      $ 1023 "barreno_actual≔barreno_actual+1"
      global barreno_actual=barreno_actual+1
    end
    $ 1026 "Popup: Linea1 con chica Terminada!"
    popup("Linea1 con chica Terminada!", "Mensaje", False, False, blocking=True)
    $ 1027 "Linea4"
    $ 1028 "Marcar_puntos"
    $ 1029 "MoveL"
    $ 1030 "punto_inicio1" "breakAfter"
    movel(punto_inicio1_p, a=0.5, v=0.1)
    $ 1031 "Linea4_A" "breakAfter"
    movel(Linea4_A_p, a=0.5, v=0.1)
    $ 1032 "Linea4_B" "breakAfter"
    movel(Linea4_B_p, a=0.5, v=0.1)
    $ 1033 "Linea4_C" "breakAfter"
    movel(Linea4_C_p, a=0.5, v=0.1)
    $ 1034 "Linea4_D" "breakAfter"
    movel(Linea4_D_p, a=0.5, v=0.1)
    $ 1035 "Linea4_E" "breakAfter"
    movel(Linea4_E_p, a=0.5, v=0.1)
    $ 1036 "Linea4_F" "breakAfter"
    movel(Linea4_F_p, a=0.5, v=0.1)
    $ 1037 "AB"
    $ 1038 "'desbaste_inicial'"
    # 'desbaste_inicial'
    $ 1039 "bajada_broca≔p[0,0,-0.012,0,0,0]"
    global bajada_broca=p[0,0,-0.012,0,0,0]
    $ 1040 "barrenos_menos1≔8"
    global barrenos_menos1=8
    $ 1041 "barreno_actual≔0"
    global barreno_actual=0
    $ 1042 "Loop barreno_actual≤barrenos_menos1"
    while (barreno_actual <= barrenos_menos1):
      $ 1043 "Perforacion"
      $ 1044 "MoveL"
      $ 1045 "internos≔interpolate_pose(Linea4_A, Linea4_B, barreno_actual/barrenos_menos1)"
      global internos= interpolate_pose (Linea4_A_p, Linea4_B_p, barreno_actual/barrenos_menos1)
      $ 1046 "internos" "breakAfter"
      movel(internos, a=0.5, v=0.1)
      $ 1047 "'desbaste_inicial'"
      # 'desbaste_inicial'
      $ 1048 "bajada_broca≔p[0,0,-0.012,0,0,0]"
      global bajada_broca=p[0,0,-0.012,0,0,0]
      $ 1049 "bajada≔p[0,0,0.012,0,0,0]"
      global bajada=p[0,0,0.012,0,0,0]
      $ 1050 "Direction: Base Z-"
      global move_thread_flag_1050=0
      thread move_thread_1050():
        enter_critical
        move_thread_flag_1050 = 1
        local towardsPos=calculate_point_to_move_towards(p[0.0,0.0,0.0,0.0,0.0,0.0], [0.0,0.0,-1.0], 0.055)
        movel(towardsPos, a=0.015, v=0.02)
        move_thread_flag_1050 = 2
        exit_critical
      end
      move_thread_flag_1050 = 0
      move_thread_han_1050 = run move_thread_1050()
      while (True):
        sleep(1.0E-10)
        if (move_thread_flag_1050 > 1):
          join move_thread_han_1050
          $ 1051 "Until (distance)"
          break
        end
        sync()
      end
      $ 1052 "Popup: punto contacto alanzdo"
      popup("punto contacto alanzdo", "Mensaje", False, False, blocking=True)
      $ 1053 "Direction: Base Z+"
      global move_thread_flag_1053=0
      thread move_thread_1053():
        enter_critical
        move_thread_flag_1053 = 1
        local towardsPos=calculate_point_to_move_towards(p[0.0,0.0,0.0,0.0,0.0,0.0], [0.0,0.0,1.0], 0.002)
        movel(towardsPos, a=0.005, v=0.003)
        move_thread_flag_1053 = 2
        exit_critical
      end
      move_thread_flag_1053 = 0
      move_thread_han_1053 = run move_thread_1053()
      while (True):
        sleep(1.0E-10)
        if (move_thread_flag_1053 > 1):
          join move_thread_han_1053
          $ 1054 "Until (distance)"
          break
        end
        sync()
      end
      $ 1055 "Wait: 0.3"
      sleep(0.3)
      $ 1056 "Set CO[1]=Encender"
      set_configurable_digital_out(1, True)
      $ 1057 "Wait: 0.3"
      sleep(0.3)
      $ 1058 "Loop 2 times"
      Loop_76 = 0
      while (Loop_76 < 2):
        $ 1059 "bajar≔pose_add(get_actual_tcp_pose(), bajada_broca)"
        global bajar= pose_add ( get_actual_tcp_pose (), bajada_broca)
        $ 1060 "bajar" "breakAfter"
        movel(bajar, a=0.005, v=0.001)
        $ 1061 "subir≔pose_sub(get_actual_tcp_pose(), bajada_broca)"
        global subir= pose_sub ( get_actual_tcp_pose (), bajada_broca)
        $ 1062 "subir" "breakAfter"
        movel(subir, a=0.01, v=0.005)
        $ 1063 "bajada_broca≔pose_sub(bajada_broca, bajada)"
        global bajada_broca= pose_sub (bajada_broca, bajada)
        Loop_76 = Loop_76 + 1
      end
      $ 1064 "Direction: Base Z+"
      global move_thread_flag_1064=0
      thread move_thread_1064():
        enter_critical
        move_thread_flag_1064 = 1
        local towardsPos=calculate_point_to_move_towards(p[0.0,0.0,0.0,0.0,0.0,0.0], [0.0,0.0,1.0], 0.06)
        movel(towardsPos, a=0.035, v=0.03)
        move_thread_flag_1064 = 2
        exit_critical
      end
      move_thread_flag_1064 = 0
      move_thread_han_1064 = run move_thread_1064()
      while (True):
        sleep(1.0E-10)
        if (move_thread_flag_1064 > 1):
          join move_thread_han_1064
          $ 1065 "Until (distance)"
          break
        end
        sync()
      end
      $ 1066 "Set CO[1]=Apagar"
      set_configurable_digital_out(1, False)
      $ 1067 "barreno_actual≔barreno_actual+1"
      global barreno_actual=barreno_actual+1
    end
    $ 1070 "CD"
    $ 1071 "'desbaste_inicial'"
    # 'desbaste_inicial'
    $ 1072 "bajada_broca≔p[0,0,-0.012,0,0,0]"
    global bajada_broca=p[0,0,-0.012,0,0,0]
    $ 1073 "barrenos_menos1≔8"
    global barrenos_menos1=8
    $ 1074 "barreno_actual≔0"
    global barreno_actual=0
    $ 1075 "Loop barreno_actual≤barrenos_menos1"
    while (barreno_actual <= barrenos_menos1):
      $ 1076 "Perforacion"
      $ 1077 "MoveL"
      $ 1078 "internos≔interpolate_pose(Linea4_C, Linea4_D, barreno_actual/barrenos_menos1)"
      global internos= interpolate_pose (Linea4_C_p, Linea4_D_p, barreno_actual/barrenos_menos1)
      $ 1079 "internos" "breakAfter"
      movel(internos, a=0.5, v=0.1)
      $ 1080 "'desbaste_inicial'"
      # 'desbaste_inicial'
      $ 1081 "bajada_broca≔p[0,0,-0.012,0,0,0]"
      global bajada_broca=p[0,0,-0.012,0,0,0]
      $ 1082 "bajada≔p[0,0,0.012,0,0,0]"
      global bajada=p[0,0,0.012,0,0,0]
      $ 1083 "Direction: Base Z-"
      global move_thread_flag_1083=0
      thread move_thread_1083():
        enter_critical
        move_thread_flag_1083 = 1
        local towardsPos=calculate_point_to_move_towards(p[0.0,0.0,0.0,0.0,0.0,0.0], [0.0,0.0,-1.0], 0.055)
        movel(towardsPos, a=0.015, v=0.02)
        move_thread_flag_1083 = 2
        exit_critical
      end
      move_thread_flag_1083 = 0
      move_thread_han_1083 = run move_thread_1083()
      while (True):
        sleep(1.0E-10)
        if (move_thread_flag_1083 > 1):
          join move_thread_han_1083
          $ 1084 "Until (distance)"
          break
        end
        sync()
      end
      $ 1085 "Popup: punto contacto alanzdo"
      popup("punto contacto alanzdo", "Mensaje", False, False, blocking=True)
      $ 1086 "Direction: Base Z+"
      global move_thread_flag_1086=0
      thread move_thread_1086():
        enter_critical
        move_thread_flag_1086 = 1
        local towardsPos=calculate_point_to_move_towards(p[0.0,0.0,0.0,0.0,0.0,0.0], [0.0,0.0,1.0], 0.002)
        movel(towardsPos, a=0.005, v=0.003)
        move_thread_flag_1086 = 2
        exit_critical
      end
      move_thread_flag_1086 = 0
      move_thread_han_1086 = run move_thread_1086()
      while (True):
        sleep(1.0E-10)
        if (move_thread_flag_1086 > 1):
          join move_thread_han_1086
          $ 1087 "Until (distance)"
          break
        end
        sync()
      end
      $ 1088 "Wait: 0.3"
      sleep(0.3)
      $ 1089 "Set CO[1]=Encender"
      set_configurable_digital_out(1, True)
      $ 1090 "Wait: 0.3"
      sleep(0.3)
      $ 1091 "Loop 2 times"
      Loop_78 = 0
      while (Loop_78 < 2):
        $ 1092 "bajar≔pose_add(get_actual_tcp_pose(), bajada_broca)"
        global bajar= pose_add ( get_actual_tcp_pose (), bajada_broca)
        $ 1093 "bajar" "breakAfter"
        movel(bajar, a=0.005, v=0.001)
        $ 1094 "subir≔pose_sub(get_actual_tcp_pose(), bajada_broca)"
        global subir= pose_sub ( get_actual_tcp_pose (), bajada_broca)
        $ 1095 "subir" "breakAfter"
        movel(subir, a=0.01, v=0.005)
        $ 1096 "bajada_broca≔pose_sub(bajada_broca, bajada)"
        global bajada_broca= pose_sub (bajada_broca, bajada)
        Loop_78 = Loop_78 + 1
      end
      $ 1097 "Direction: Base Z+"
      global move_thread_flag_1097=0
      thread move_thread_1097():
        enter_critical
        move_thread_flag_1097 = 1
        local towardsPos=calculate_point_to_move_towards(p[0.0,0.0,0.0,0.0,0.0,0.0], [0.0,0.0,1.0], 0.06)
        movel(towardsPos, a=0.035, v=0.03)
        move_thread_flag_1097 = 2
        exit_critical
      end
      move_thread_flag_1097 = 0
      move_thread_han_1097 = run move_thread_1097()
      while (True):
        sleep(1.0E-10)
        if (move_thread_flag_1097 > 1):
          join move_thread_han_1097
          $ 1098 "Until (distance)"
          break
        end
        sync()
      end
      $ 1099 "Set CO[1]=Apagar"
      set_configurable_digital_out(1, False)
      $ 1100 "barreno_actual≔barreno_actual+1"
      global barreno_actual=barreno_actual+1
    end
    $ 1103 "EF"
    $ 1104 "'desbaste_inicial'"
    # 'desbaste_inicial'
    $ 1105 "bajada_broca≔p[0,0,-0.012,0,0,0]"
    global bajada_broca=p[0,0,-0.012,0,0,0]
    $ 1106 "barrenos_menos1≔9"
    global barrenos_menos1=9
    $ 1107 "barreno_actual≔0"
    global barreno_actual=0
    $ 1108 "Loop barreno_actual≤barrenos_menos1"
    while (barreno_actual <= barrenos_menos1):
      $ 1109 "Perforacion"
      $ 1110 "MoveL"
      $ 1111 "internos≔interpolate_pose(Linea4_E, Linea4_F, barreno_actual/barrenos_menos1)"
      global internos= interpolate_pose (Linea4_E_p, Linea4_F_p, barreno_actual/barrenos_menos1)
      $ 1112 "internos" "breakAfter"
      movel(internos, a=0.5, v=0.1)
      $ 1113 "'desbaste_inicial'"
      # 'desbaste_inicial'
      $ 1114 "bajada_broca≔p[0,0,-0.012,0,0,0]"
      global bajada_broca=p[0,0,-0.012,0,0,0]
      $ 1115 "bajada≔p[0,0,0.012,0,0,0]"
      global bajada=p[0,0,0.012,0,0,0]
      $ 1116 "Direction: Base Z-"
      global move_thread_flag_1116=0
      thread move_thread_1116():
        enter_critical
        move_thread_flag_1116 = 1
        local towardsPos=calculate_point_to_move_towards(p[0.0,0.0,0.0,0.0,0.0,0.0], [0.0,0.0,-1.0], 0.055)
        movel(towardsPos, a=0.015, v=0.02)
        move_thread_flag_1116 = 2
        exit_critical
      end
      move_thread_flag_1116 = 0
      move_thread_han_1116 = run move_thread_1116()
      while (True):
        sleep(1.0E-10)
        if (move_thread_flag_1116 > 1):
          join move_thread_han_1116
          $ 1117 "Until (distance)"
          break
        end
        sync()
      end
      $ 1118 "Popup: punto contacto alanzdo"
      popup("punto contacto alanzdo", "Mensaje", False, False, blocking=True)
      $ 1119 "Direction: Base Z+"
      global move_thread_flag_1119=0
      thread move_thread_1119():
        enter_critical
        move_thread_flag_1119 = 1
        local towardsPos=calculate_point_to_move_towards(p[0.0,0.0,0.0,0.0,0.0,0.0], [0.0,0.0,1.0], 0.002)
        movel(towardsPos, a=0.005, v=0.003)
        move_thread_flag_1119 = 2
        exit_critical
      end
      move_thread_flag_1119 = 0
      move_thread_han_1119 = run move_thread_1119()
      while (True):
        sleep(1.0E-10)
        if (move_thread_flag_1119 > 1):
          join move_thread_han_1119
          $ 1120 "Until (distance)"
          break
        end
        sync()
      end
      $ 1121 "Wait: 0.3"
      sleep(0.3)
      $ 1122 "Set CO[1]=Encender"
      set_configurable_digital_out(1, True)
      $ 1123 "Wait: 0.3"
      sleep(0.3)
      $ 1124 "Loop 2 times"
      Loop_80 = 0
      while (Loop_80 < 2):
        $ 1125 "bajar≔pose_add(get_actual_tcp_pose(), bajada_broca)"
        global bajar= pose_add ( get_actual_tcp_pose (), bajada_broca)
        $ 1126 "bajar" "breakAfter"
        movel(bajar, a=0.005, v=0.001)
        $ 1127 "subir≔pose_sub(get_actual_tcp_pose(), bajada_broca)"
        global subir= pose_sub ( get_actual_tcp_pose (), bajada_broca)
        $ 1128 "subir" "breakAfter"
        movel(subir, a=0.01, v=0.005)
        $ 1129 "bajada_broca≔pose_sub(bajada_broca, bajada)"
        global bajada_broca= pose_sub (bajada_broca, bajada)
        Loop_80 = Loop_80 + 1
      end
      $ 1130 "Direction: Base Z+"
      global move_thread_flag_1130=0
      thread move_thread_1130():
        enter_critical
        move_thread_flag_1130 = 1
        local towardsPos=calculate_point_to_move_towards(p[0.0,0.0,0.0,0.0,0.0,0.0], [0.0,0.0,1.0], 0.06)
        movel(towardsPos, a=0.035, v=0.03)
        move_thread_flag_1130 = 2
        exit_critical
      end
      move_thread_flag_1130 = 0
      move_thread_han_1130 = run move_thread_1130()
      while (True):
        sleep(1.0E-10)
        if (move_thread_flag_1130 > 1):
          join move_thread_han_1130
          $ 1131 "Until (distance)"
          break
        end
        sync()
      end
      $ 1132 "Set CO[1]=Apagar"
      set_configurable_digital_out(1, False)
      $ 1133 "barreno_actual≔barreno_actual+1"
      global barreno_actual=barreno_actual+1
      $ 1134 "If barreno_actual>barrenos_menos1"
      if (barreno_actual>barrenos_menos1):
        $ 1135 "cambiar_broca≔ True "
        global cambiar_broca=  True
      end
    end
    $ 1138 "Popup: Linea2 con chica Terminada!"
    popup("Linea2 con chica Terminada!", "Mensaje", False, False, blocking=True)
    $ 1139 "Broca_3"
    $ 1140 "Linea3"
    $ 1141 "Marcar_puntos"
    $ 1142 "MoveL"
    $ 1143 "punto_inicio1" "breakAfter"
    movel(punto_inicio1_p, a=0.5, v=0.1)
    $ 1144 "Linea3_A" "breakAfter"
    movel(Linea3_A_p, a=0.5, v=0.1)
    $ 1145 "Linea3_B" "breakAfter"
    movel(Linea3_B_p, a=0.5, v=0.1)
    $ 1146 "Linea3_C" "breakAfter"
    movel(Linea3_C_p, a=0.5, v=0.1)
    $ 1147 "Linea3_D" "breakAfter"
    movel(Linea3_D_p, a=0.5, v=0.1)
    $ 1148 "Linea3_E" "breakAfter"
    movel(Linea3_E_p, a=0.5, v=0.1)
    $ 1149 "Linea3_F" "breakAfter"
    movel(Linea3_F_p, a=0.5, v=0.1)
    $ 1150 "AB"
    $ 1151 "'desbaste_inicial'"
    # 'desbaste_inicial'
    $ 1152 "bajada_broca≔p[0,0,-0.012,0,0,0]"
    global bajada_broca=p[0,0,-0.012,0,0,0]
    $ 1153 "barrenos_menos1≔8"
    global barrenos_menos1=8
    $ 1154 "barreno_actual≔0"
    global barreno_actual=0
    $ 1155 "Loop barreno_actual≤barrenos_menos1"
    while (barreno_actual <= barrenos_menos1):
      $ 1156 "Perforacion"
      $ 1157 "MoveL"
      $ 1158 "internos≔interpolate_pose(Linea3_A, Linea3_B, barreno_actual/barrenos_menos1)"
      global internos= interpolate_pose (Linea3_A_p, Linea3_B_p, barreno_actual/barrenos_menos1)
      $ 1159 "internos" "breakAfter"
      movel(internos, a=0.5, v=0.1)
      $ 1160 "'desbaste_inicial'"
      # 'desbaste_inicial'
      $ 1161 "bajada_broca≔p[0,0,-0.012,0,0,0]"
      global bajada_broca=p[0,0,-0.012,0,0,0]
      $ 1162 "bajada≔p[0,0,0.012,0,0,0]"
      global bajada=p[0,0,0.012,0,0,0]
      $ 1163 "Direction: Base Z-"
      global move_thread_flag_1163=0
      thread move_thread_1163():
        enter_critical
        move_thread_flag_1163 = 1
        local towardsPos=calculate_point_to_move_towards(p[0.0,0.0,0.0,0.0,0.0,0.0], [0.0,0.0,-1.0], 0.06)
        movel(towardsPos, a=0.015, v=0.02)
        move_thread_flag_1163 = 2
        exit_critical
      end
      move_thread_flag_1163 = 0
      move_thread_han_1163 = run move_thread_1163()
      while (True):
        sleep(1.0E-10)
        if (move_thread_flag_1163 > 1):
          join move_thread_han_1163
          $ 1164 "Until (distance)"
          break
        end
        sync()
      end
      $ 1165 "Popup: punto contacto alanzdo"
      popup("punto contacto alanzdo", "Mensaje", False, False, blocking=True)
      $ 1166 "Direction: Base Z+"
      global move_thread_flag_1166=0
      thread move_thread_1166():
        enter_critical
        move_thread_flag_1166 = 1
        local towardsPos=calculate_point_to_move_towards(p[0.0,0.0,0.0,0.0,0.0,0.0], [0.0,0.0,1.0], 0.002)
        movel(towardsPos, a=0.005, v=0.003)
        move_thread_flag_1166 = 2
        exit_critical
      end
      move_thread_flag_1166 = 0
      move_thread_han_1166 = run move_thread_1166()
      while (True):
        sleep(1.0E-10)
        if (move_thread_flag_1166 > 1):
          join move_thread_han_1166
          $ 1167 "Until (distance)"
          break
        end
        sync()
      end
      $ 1168 "Wait: 0.3"
      sleep(0.3)
      $ 1169 "Set CO[1]=Encender"
      set_configurable_digital_out(1, True)
      $ 1170 "Wait: 0.3"
      sleep(0.3)
      $ 1171 "Loop 2 times"
      Loop_82 = 0
      while (Loop_82 < 2):
        $ 1172 "bajar≔pose_add(get_actual_tcp_pose(), bajada_broca)"
        global bajar= pose_add ( get_actual_tcp_pose (), bajada_broca)
        $ 1173 "bajar" "breakAfter"
        movel(bajar, a=0.005, v=0.001)
        $ 1174 "subir≔pose_sub(get_actual_tcp_pose(), bajada_broca)"
        global subir= pose_sub ( get_actual_tcp_pose (), bajada_broca)
        $ 1175 "subir" "breakAfter"
        movel(subir, a=0.01, v=0.01)
        $ 1176 "bajada_broca≔pose_sub(bajada_broca, bajada)"
        global bajada_broca= pose_sub (bajada_broca, bajada)
        Loop_82 = Loop_82 + 1
      end
      $ 1177 "Direction: Base Z+"
      global move_thread_flag_1177=0
      thread move_thread_1177():
        enter_critical
        move_thread_flag_1177 = 1
        local towardsPos=calculate_point_to_move_towards(p[0.0,0.0,0.0,0.0,0.0,0.0], [0.0,0.0,1.0], 0.06)
        movel(towardsPos, a=0.035, v=0.03)
        move_thread_flag_1177 = 2
        exit_critical
      end
      move_thread_flag_1177 = 0
      move_thread_han_1177 = run move_thread_1177()
      while (True):
        sleep(1.0E-10)
        if (move_thread_flag_1177 > 1):
          join move_thread_han_1177
          $ 1178 "Until (distance)"
          break
        end
        sync()
      end
      $ 1179 "Set CO[1]=Apagar"
      set_configurable_digital_out(1, False)
      $ 1180 "barreno_actual≔barreno_actual+1"
      global barreno_actual=barreno_actual+1
    end
    $ 1183 "CD"
    $ 1184 "'desbaste_inicial'"
    # 'desbaste_inicial'
    $ 1185 "bajada_broca≔p[0,0,-0.012,0,0,0]"
    global bajada_broca=p[0,0,-0.012,0,0,0]
    $ 1186 "barrenos_menos1≔8"
    global barrenos_menos1=8
    $ 1187 "barreno_actual≔0"
    global barreno_actual=0
    $ 1188 "Loop barreno_actual≤barrenos_menos1"
    while (barreno_actual <= barrenos_menos1):
      $ 1189 "Perforacion"
      $ 1190 "MoveL"
      $ 1191 "internos≔interpolate_pose(Linea3_C, Linea3_D, barreno_actual/barrenos_menos1)"
      global internos= interpolate_pose (Linea3_C_p, Linea3_D_p, barreno_actual/barrenos_menos1)
      $ 1192 "internos" "breakAfter"
      movel(internos, a=0.5, v=0.1)
      $ 1193 "'desbaste_inicial'"
      # 'desbaste_inicial'
      $ 1194 "bajada_broca≔p[0,0,-0.012,0,0,0]"
      global bajada_broca=p[0,0,-0.012,0,0,0]
      $ 1195 "bajada≔p[0,0,0.012,0,0,0]"
      global bajada=p[0,0,0.012,0,0,0]
      $ 1196 "Direction: Base Z-"
      global move_thread_flag_1196=0
      thread move_thread_1196():
        enter_critical
        move_thread_flag_1196 = 1
        local towardsPos=calculate_point_to_move_towards(p[0.0,0.0,0.0,0.0,0.0,0.0], [0.0,0.0,-1.0], 0.06)
        movel(towardsPos, a=0.02, v=0.015)
        move_thread_flag_1196 = 2
        exit_critical
      end
      move_thread_flag_1196 = 0
      move_thread_han_1196 = run move_thread_1196()
      while (True):
        sleep(1.0E-10)
        if (move_thread_flag_1196 > 1):
          join move_thread_han_1196
          $ 1197 "Until (distance)"
          break
        end
        sync()
      end
      $ 1198 "Popup: punto contacto alanzdo"
      popup("punto contacto alanzdo", "Mensaje", False, False, blocking=True)
      $ 1199 "Direction: Base Z+"
      global move_thread_flag_1199=0
      thread move_thread_1199():
        enter_critical
        move_thread_flag_1199 = 1
        local towardsPos=calculate_point_to_move_towards(p[0.0,0.0,0.0,0.0,0.0,0.0], [0.0,0.0,1.0], 0.002)
        movel(towardsPos, a=0.005, v=0.003)
        move_thread_flag_1199 = 2
        exit_critical
      end
      move_thread_flag_1199 = 0
      move_thread_han_1199 = run move_thread_1199()
      while (True):
        sleep(1.0E-10)
        if (move_thread_flag_1199 > 1):
          join move_thread_han_1199
          $ 1200 "Until (distance)"
          break
        end
        sync()
      end
      $ 1201 "Wait: 0.3"
      sleep(0.3)
      $ 1202 "Set CO[1]=Encender"
      set_configurable_digital_out(1, True)
      $ 1203 "Wait: 0.3"
      sleep(0.3)
      $ 1204 "Loop 2 times"
      Loop_84 = 0
      while (Loop_84 < 2):
        $ 1205 "bajar≔pose_add(get_actual_tcp_pose(), bajada_broca)"
        global bajar= pose_add ( get_actual_tcp_pose (), bajada_broca)
        $ 1206 "bajar" "breakAfter"
        movel(bajar, a=0.005, v=0.001)
        $ 1207 "subir≔pose_sub(get_actual_tcp_pose(), bajada_broca)"
        global subir= pose_sub ( get_actual_tcp_pose (), bajada_broca)
        $ 1208 "subir" "breakAfter"
        movel(subir, a=0.01, v=0.01)
        $ 1209 "bajada_broca≔pose_sub(bajada_broca, bajada)"
        global bajada_broca= pose_sub (bajada_broca, bajada)
        Loop_84 = Loop_84 + 1
      end
      $ 1210 "Direction: Base Z+"
      global move_thread_flag_1210=0
      thread move_thread_1210():
        enter_critical
        move_thread_flag_1210 = 1
        local towardsPos=calculate_point_to_move_towards(p[0.0,0.0,0.0,0.0,0.0,0.0], [0.0,0.0,1.0], 0.06)
        movel(towardsPos, a=0.035, v=0.03)
        move_thread_flag_1210 = 2
        exit_critical
      end
      move_thread_flag_1210 = 0
      move_thread_han_1210 = run move_thread_1210()
      while (True):
        sleep(1.0E-10)
        if (move_thread_flag_1210 > 1):
          join move_thread_han_1210
          $ 1211 "Until (distance)"
          break
        end
        sync()
      end
      $ 1212 "Set CO[1]=Apagar"
      set_configurable_digital_out(1, False)
      $ 1213 "barreno_actual≔barreno_actual+1"
      global barreno_actual=barreno_actual+1
    end
    $ 1216 "EF"
    $ 1217 "'desbaste_inicial'"
    # 'desbaste_inicial'
    $ 1218 "bajada_broca≔p[0,0,-0.012,0,0,0]"
    global bajada_broca=p[0,0,-0.012,0,0,0]
    $ 1219 "barrenos_menos1≔9"
    global barrenos_menos1=9
    $ 1220 "barreno_actual≔0"
    global barreno_actual=0
    $ 1221 "Loop barreno_actual≤barrenos_menos1"
    while (barreno_actual <= barrenos_menos1):
      $ 1222 "Perforacion"
      $ 1223 "MoveL"
      $ 1224 "internos≔interpolate_pose(Linea3_E, Linea3_F, barreno_actual/barrenos_menos1)"
      global internos= interpolate_pose (Linea3_E_p, Linea3_F_p, barreno_actual/barrenos_menos1)
      $ 1225 "internos" "breakAfter"
      movel(internos, a=0.5, v=0.1)
      $ 1226 "'desbaste_inicial'"
      # 'desbaste_inicial'
      $ 1227 "bajada_broca≔p[0,0,-0.012,0,0,0]"
      global bajada_broca=p[0,0,-0.012,0,0,0]
      $ 1228 "bajada≔p[0,0,0.012,0,0,0]"
      global bajada=p[0,0,0.012,0,0,0]
      $ 1229 "Direction: Base Z-"
      global move_thread_flag_1229=0
      thread move_thread_1229():
        enter_critical
        move_thread_flag_1229 = 1
        local towardsPos=calculate_point_to_move_towards(p[0.0,0.0,0.0,0.0,0.0,0.0], [0.0,0.0,-1.0], 0.06)
        movel(towardsPos, a=0.015, v=0.02)
        move_thread_flag_1229 = 2
        exit_critical
      end
      move_thread_flag_1229 = 0
      move_thread_han_1229 = run move_thread_1229()
      while (True):
        sleep(1.0E-10)
        if (move_thread_flag_1229 > 1):
          join move_thread_han_1229
          $ 1230 "Until (distance)"
          break
        end
        sync()
      end
      $ 1231 "Popup: punto contacto alanzdo"
      popup("punto contacto alanzdo", "Mensaje", False, False, blocking=True)
      $ 1232 "Direction: Base Z+"
      global move_thread_flag_1232=0
      thread move_thread_1232():
        enter_critical
        move_thread_flag_1232 = 1
        local towardsPos=calculate_point_to_move_towards(p[0.0,0.0,0.0,0.0,0.0,0.0], [0.0,0.0,1.0], 0.002)
        movel(towardsPos, a=0.005, v=0.003)
        move_thread_flag_1232 = 2
        exit_critical
      end
      move_thread_flag_1232 = 0
      move_thread_han_1232 = run move_thread_1232()
      while (True):
        sleep(1.0E-10)
        if (move_thread_flag_1232 > 1):
          join move_thread_han_1232
          $ 1233 "Until (distance)"
          break
        end
        sync()
      end
      $ 1234 "Wait: 0.3"
      sleep(0.3)
      $ 1235 "Set CO[1]=Encender"
      set_configurable_digital_out(1, True)
      $ 1236 "Wait: 0.3"
      sleep(0.3)
      $ 1237 "Loop 2 times"
      Loop_86 = 0
      while (Loop_86 < 2):
        $ 1238 "bajar≔pose_add(get_actual_tcp_pose(), bajada_broca)"
        global bajar= pose_add ( get_actual_tcp_pose (), bajada_broca)
        $ 1239 "bajar" "breakAfter"
        movel(bajar, a=0.005, v=0.001)
        $ 1240 "subir≔pose_sub(get_actual_tcp_pose(), bajada_broca)"
        global subir= pose_sub ( get_actual_tcp_pose (), bajada_broca)
        $ 1241 "subir" "breakAfter"
        movel(subir, a=0.01, v=0.01)
        $ 1242 "bajada_broca≔pose_sub(bajada_broca, bajada)"
        global bajada_broca= pose_sub (bajada_broca, bajada)
        Loop_86 = Loop_86 + 1
      end
      $ 1243 "Direction: Base Z+"
      global move_thread_flag_1243=0
      thread move_thread_1243():
        enter_critical
        move_thread_flag_1243 = 1
        local towardsPos=calculate_point_to_move_towards(p[0.0,0.0,0.0,0.0,0.0,0.0], [0.0,0.0,1.0], 0.06)
        movel(towardsPos, a=0.035, v=0.03)
        move_thread_flag_1243 = 2
        exit_critical
      end
      move_thread_flag_1243 = 0
      move_thread_han_1243 = run move_thread_1243()
      while (True):
        sleep(1.0E-10)
        if (move_thread_flag_1243 > 1):
          join move_thread_han_1243
          $ 1244 "Until (distance)"
          break
        end
        sync()
      end
      $ 1245 "Set CO[1]=Apagar"
      set_configurable_digital_out(1, False)
      $ 1246 "barreno_actual≔barreno_actual+1"
      global barreno_actual=barreno_actual+1
    end
    $ 1249 "Popup: Linea1 con chica Terminada!"
    popup("Linea1 con chica Terminada!", "Mensaje", False, False, blocking=True)
    $ 1250 "Linea4"
    $ 1251 "Marcar_puntos"
    $ 1252 "MoveL"
    $ 1253 "punto_inicio1" "breakAfter"
    movel(punto_inicio1_p, a=0.5, v=0.1)
    $ 1254 "Linea4_A" "breakAfter"
    movel(Linea4_A_p, a=0.5, v=0.1)
    $ 1255 "Linea4_B" "breakAfter"
    movel(Linea4_B_p, a=0.5, v=0.1)
    $ 1256 "Linea4_C" "breakAfter"
    movel(Linea4_C_p, a=0.5, v=0.1)
    $ 1257 "Linea4_D" "breakAfter"
    movel(Linea4_D_p, a=0.5, v=0.1)
    $ 1258 "Linea4_E" "breakAfter"
    movel(Linea4_E_p, a=0.5, v=0.1)
    $ 1259 "Linea4_F" "breakAfter"
    movel(Linea4_F_p, a=0.5, v=0.1)
    $ 1260 "AB"
    $ 1261 "'desbaste_inicial'"
    # 'desbaste_inicial'
    $ 1262 "bajada_broca≔p[0,0,-0.012,0,0,0]"
    global bajada_broca=p[0,0,-0.012,0,0,0]
    $ 1263 "barrenos_menos1≔8"
    global barrenos_menos1=8
    $ 1264 "barreno_actual≔0"
    global barreno_actual=0
    $ 1265 "Loop barreno_actual≤barrenos_menos1"
    while (barreno_actual <= barrenos_menos1):
      $ 1266 "Perforacion"
      $ 1267 "MoveL"
      $ 1268 "internos≔interpolate_pose(Linea4_A, Linea4_B, barreno_actual/barrenos_menos1)"
      global internos= interpolate_pose (Linea4_A_p, Linea4_B_p, barreno_actual/barrenos_menos1)
      $ 1269 "internos" "breakAfter"
      movel(internos, a=0.5, v=0.1)
      $ 1270 "'desbaste_inicial'"
      # 'desbaste_inicial'
      $ 1271 "bajada_broca≔p[0,0,-0.012,0,0,0]"
      global bajada_broca=p[0,0,-0.012,0,0,0]
      $ 1272 "bajada≔p[0,0,0.012,0,0,0]"
      global bajada=p[0,0,0.012,0,0,0]
      $ 1273 "Direction: Base Z-"
      global move_thread_flag_1273=0
      thread move_thread_1273():
        enter_critical
        move_thread_flag_1273 = 1
        local towardsPos=calculate_point_to_move_towards(p[0.0,0.0,0.0,0.0,0.0,0.0], [0.0,0.0,-1.0], 0.06)
        movel(towardsPos, a=0.015, v=0.02)
        move_thread_flag_1273 = 2
        exit_critical
      end
      move_thread_flag_1273 = 0
      move_thread_han_1273 = run move_thread_1273()
      while (True):
        sleep(1.0E-10)
        if (move_thread_flag_1273 > 1):
          join move_thread_han_1273
          $ 1274 "Until (distance)"
          break
        end
        sync()
      end
      $ 1275 "Popup: punto contacto alanzdo"
      popup("punto contacto alanzdo", "Mensaje", False, False, blocking=True)
      $ 1276 "Direction: Base Z+"
      global move_thread_flag_1276=0
      thread move_thread_1276():
        enter_critical
        move_thread_flag_1276 = 1
        local towardsPos=calculate_point_to_move_towards(p[0.0,0.0,0.0,0.0,0.0,0.0], [0.0,0.0,1.0], 0.002)
        movel(towardsPos, a=0.005, v=0.003)
        move_thread_flag_1276 = 2
        exit_critical
      end
      move_thread_flag_1276 = 0
      move_thread_han_1276 = run move_thread_1276()
      while (True):
        sleep(1.0E-10)
        if (move_thread_flag_1276 > 1):
          join move_thread_han_1276
          $ 1277 "Until (distance)"
          break
        end
        sync()
      end
      $ 1278 "Wait: 0.3"
      sleep(0.3)
      $ 1279 "Set CO[1]=Encender"
      set_configurable_digital_out(1, True)
      $ 1280 "Wait: 0.3"
      sleep(0.3)
      $ 1281 "Loop 2 times"
      Loop_88 = 0
      while (Loop_88 < 2):
        $ 1282 "bajar≔pose_add(get_actual_tcp_pose(), bajada_broca)"
        global bajar= pose_add ( get_actual_tcp_pose (), bajada_broca)
        $ 1283 "bajar" "breakAfter"
        movel(bajar, a=0.005, v=0.001)
        $ 1284 "subir≔pose_sub(get_actual_tcp_pose(), bajada_broca)"
        global subir= pose_sub ( get_actual_tcp_pose (), bajada_broca)
        $ 1285 "subir" "breakAfter"
        movel(subir, a=0.01, v=0.01)
        $ 1286 "bajada_broca≔pose_sub(bajada_broca, bajada)"
        global bajada_broca= pose_sub (bajada_broca, bajada)
        Loop_88 = Loop_88 + 1
      end
      $ 1287 "Direction: Base Z+"
      global move_thread_flag_1287=0
      thread move_thread_1287():
        enter_critical
        move_thread_flag_1287 = 1
        local towardsPos=calculate_point_to_move_towards(p[0.0,0.0,0.0,0.0,0.0,0.0], [0.0,0.0,1.0], 0.06)
        movel(towardsPos, a=0.035, v=0.03)
        move_thread_flag_1287 = 2
        exit_critical
      end
      move_thread_flag_1287 = 0
      move_thread_han_1287 = run move_thread_1287()
      while (True):
        sleep(1.0E-10)
        if (move_thread_flag_1287 > 1):
          join move_thread_han_1287
          $ 1288 "Until (distance)"
          break
        end
        sync()
      end
      $ 1289 "Set CO[1]=Apagar"
      set_configurable_digital_out(1, False)
      $ 1290 "barreno_actual≔barreno_actual+1"
      global barreno_actual=barreno_actual+1
    end
    $ 1293 "CD"
    $ 1294 "'desbaste_inicial'"
    # 'desbaste_inicial'
    $ 1295 "bajada_broca≔p[0,0,-0.012,0,0,0]"
    global bajada_broca=p[0,0,-0.012,0,0,0]
    $ 1296 "barrenos_menos1≔8"
    global barrenos_menos1=8
    $ 1297 "barreno_actual≔0"
    global barreno_actual=0
    $ 1298 "Loop barreno_actual≤barrenos_menos1"
    while (barreno_actual <= barrenos_menos1):
      $ 1299 "Perforacion"
      $ 1300 "MoveL"
      $ 1301 "internos≔interpolate_pose(Linea4_C, Linea4_D, barreno_actual/barrenos_menos1)"
      global internos= interpolate_pose (Linea4_C_p, Linea4_D_p, barreno_actual/barrenos_menos1)
      $ 1302 "internos" "breakAfter"
      movel(internos, a=0.5, v=0.1)
      $ 1303 "'desbaste_inicial'"
      # 'desbaste_inicial'
      $ 1304 "bajada_broca≔p[0,0,-0.012,0,0,0]"
      global bajada_broca=p[0,0,-0.012,0,0,0]
      $ 1305 "bajada≔p[0,0,0.012,0,0,0]"
      global bajada=p[0,0,0.012,0,0,0]
      $ 1306 "Direction: Base Z-"
      global move_thread_flag_1306=0
      thread move_thread_1306():
        enter_critical
        move_thread_flag_1306 = 1
        local towardsPos=calculate_point_to_move_towards(p[0.0,0.0,0.0,0.0,0.0,0.0], [0.0,0.0,-1.0], 0.06)
        movel(towardsPos, a=0.015, v=0.02)
        move_thread_flag_1306 = 2
        exit_critical
      end
      move_thread_flag_1306 = 0
      move_thread_han_1306 = run move_thread_1306()
      while (True):
        sleep(1.0E-10)
        if (move_thread_flag_1306 > 1):
          join move_thread_han_1306
          $ 1307 "Until (distance)"
          break
        end
        sync()
      end
      $ 1308 "Popup: punto contacto alanzdo"
      popup("punto contacto alanzdo", "Mensaje", False, False, blocking=True)
      $ 1309 "Direction: Base Z+"
      global move_thread_flag_1309=0
      thread move_thread_1309():
        enter_critical
        move_thread_flag_1309 = 1
        local towardsPos=calculate_point_to_move_towards(p[0.0,0.0,0.0,0.0,0.0,0.0], [0.0,0.0,1.0], 0.002)
        movel(towardsPos, a=0.005, v=0.003)
        move_thread_flag_1309 = 2
        exit_critical
      end
      move_thread_flag_1309 = 0
      move_thread_han_1309 = run move_thread_1309()
      while (True):
        sleep(1.0E-10)
        if (move_thread_flag_1309 > 1):
          join move_thread_han_1309
          $ 1310 "Until (distance)"
          break
        end
        sync()
      end
      $ 1311 "Wait: 0.3"
      sleep(0.3)
      $ 1312 "Set CO[1]=Encender"
      set_configurable_digital_out(1, True)
      $ 1313 "Wait: 0.3"
      sleep(0.3)
      $ 1314 "Loop 2 times"
      Loop_90 = 0
      while (Loop_90 < 2):
        $ 1315 "bajar≔pose_add(get_actual_tcp_pose(), bajada_broca)"
        global bajar= pose_add ( get_actual_tcp_pose (), bajada_broca)
        $ 1316 "bajar" "breakAfter"
        movel(bajar, a=0.005, v=0.001)
        $ 1317 "subir≔pose_sub(get_actual_tcp_pose(), bajada_broca)"
        global subir= pose_sub ( get_actual_tcp_pose (), bajada_broca)
        $ 1318 "subir" "breakAfter"
        movel(subir, a=0.01, v=0.01)
        $ 1319 "bajada_broca≔pose_sub(bajada_broca, bajada)"
        global bajada_broca= pose_sub (bajada_broca, bajada)
        Loop_90 = Loop_90 + 1
      end
      $ 1320 "Direction: Base Z+"
      global move_thread_flag_1320=0
      thread move_thread_1320():
        enter_critical
        move_thread_flag_1320 = 1
        local towardsPos=calculate_point_to_move_towards(p[0.0,0.0,0.0,0.0,0.0,0.0], [0.0,0.0,1.0], 0.06)
        movel(towardsPos, a=0.035, v=0.03)
        move_thread_flag_1320 = 2
        exit_critical
      end
      move_thread_flag_1320 = 0
      move_thread_han_1320 = run move_thread_1320()
      while (True):
        sleep(1.0E-10)
        if (move_thread_flag_1320 > 1):
          join move_thread_han_1320
          $ 1321 "Until (distance)"
          break
        end
        sync()
      end
      $ 1322 "Set CO[1]=Apagar"
      set_configurable_digital_out(1, False)
      $ 1323 "barreno_actual≔barreno_actual+1"
      global barreno_actual=barreno_actual+1
    end
    $ 1326 "EF"
    $ 1327 "'desbaste_inicial'"
    # 'desbaste_inicial'
    $ 1328 "bajada_broca≔p[0,0,-0.012,0,0,0]"
    global bajada_broca=p[0,0,-0.012,0,0,0]
    $ 1329 "barrenos_menos1≔9"
    global barrenos_menos1=9
    $ 1330 "barreno_actual≔0"
    global barreno_actual=0
    $ 1331 "Loop barreno_actual≤barrenos_menos1"
    while (barreno_actual <= barrenos_menos1):
      $ 1332 "Perforacion"
      $ 1333 "MoveL"
      $ 1334 "internos≔interpolate_pose(Linea4_E, Linea4_F, barreno_actual/barrenos_menos1)"
      global internos= interpolate_pose (Linea4_E_p, Linea4_F_p, barreno_actual/barrenos_menos1)
      $ 1335 "internos" "breakAfter"
      movel(internos, a=0.5, v=0.1)
      $ 1336 "'desbaste_inicial'"
      # 'desbaste_inicial'
      $ 1337 "bajada_broca≔p[0,0,-0.012,0,0,0]"
      global bajada_broca=p[0,0,-0.012,0,0,0]
      $ 1338 "bajada≔p[0,0,0.012,0,0,0]"
      global bajada=p[0,0,0.012,0,0,0]
      $ 1339 "Direction: Base Z-"
      global move_thread_flag_1339=0
      thread move_thread_1339():
        enter_critical
        move_thread_flag_1339 = 1
        local towardsPos=calculate_point_to_move_towards(p[0.0,0.0,0.0,0.0,0.0,0.0], [0.0,0.0,-1.0], 0.06)
        movel(towardsPos, a=0.015, v=0.02)
        move_thread_flag_1339 = 2
        exit_critical
      end
      move_thread_flag_1339 = 0
      move_thread_han_1339 = run move_thread_1339()
      while (True):
        sleep(1.0E-10)
        if (move_thread_flag_1339 > 1):
          join move_thread_han_1339
          $ 1340 "Until (distance)"
          break
        end
        sync()
      end
      $ 1341 "Popup: punto contacto alanzdo"
      popup("punto contacto alanzdo", "Mensaje", False, False, blocking=True)
      $ 1342 "Direction: Base Z+"
      global move_thread_flag_1342=0
      thread move_thread_1342():
        enter_critical
        move_thread_flag_1342 = 1
        local towardsPos=calculate_point_to_move_towards(p[0.0,0.0,0.0,0.0,0.0,0.0], [0.0,0.0,1.0], 0.002)
        movel(towardsPos, a=0.005, v=0.003)
        move_thread_flag_1342 = 2
        exit_critical
      end
      move_thread_flag_1342 = 0
      move_thread_han_1342 = run move_thread_1342()
      while (True):
        sleep(1.0E-10)
        if (move_thread_flag_1342 > 1):
          join move_thread_han_1342
          $ 1343 "Until (distance)"
          break
        end
        sync()
      end
      $ 1344 "Wait: 0.3"
      sleep(0.3)
      $ 1345 "Set CO[1]=Encender"
      set_configurable_digital_out(1, True)
      $ 1346 "Wait: 0.3"
      sleep(0.3)
      $ 1347 "Loop 2 times"
      Loop_92 = 0
      while (Loop_92 < 2):
        $ 1348 "bajar≔pose_add(get_actual_tcp_pose(), bajada_broca)"
        global bajar= pose_add ( get_actual_tcp_pose (), bajada_broca)
        $ 1349 "bajar" "breakAfter"
        movel(bajar, a=0.005, v=0.001)
        $ 1350 "subir≔pose_sub(get_actual_tcp_pose(), bajada_broca)"
        global subir= pose_sub ( get_actual_tcp_pose (), bajada_broca)
        $ 1351 "subir" "breakAfter"
        movel(subir, a=0.01, v=0.01)
        $ 1352 "bajada_broca≔pose_sub(bajada_broca, bajada)"
        global bajada_broca= pose_sub (bajada_broca, bajada)
        Loop_92 = Loop_92 + 1
      end
      $ 1353 "Direction: Base Z+"
      global move_thread_flag_1353=0
      thread move_thread_1353():
        enter_critical
        move_thread_flag_1353 = 1
        local towardsPos=calculate_point_to_move_towards(p[0.0,0.0,0.0,0.0,0.0,0.0], [0.0,0.0,1.0], 0.06)
        movel(towardsPos, a=0.035, v=0.03)
        move_thread_flag_1353 = 2
        exit_critical
      end
      move_thread_flag_1353 = 0
      move_thread_han_1353 = run move_thread_1353()
      while (True):
        sleep(1.0E-10)
        if (move_thread_flag_1353 > 1):
          join move_thread_han_1353
          $ 1354 "Until (distance)"
          break
        end
        sync()
      end
      $ 1355 "Set CO[1]=Apagar"
      set_configurable_digital_out(1, False)
      $ 1356 "barreno_actual≔barreno_actual+1"
      global barreno_actual=barreno_actual+1
      $ 1357 "If barreno_actual>barrenos_menos1"
      if (barreno_actual>barrenos_menos1):
        $ 1358 "cambiar_broca≔ True "
        global cambiar_broca=  True
      end
    end
    $ 1361 "Popup: Linea2 con chica Terminada!"
    popup("Linea2 con chica Terminada!", "Mensaje", False, False, blocking=True)
    $ 1808 "'Subprogramas:'"
    # 'Subprogramas:'
  end
end
